FUNCTION_BLOCK Section1
  (* Standard: 61499-2 *)
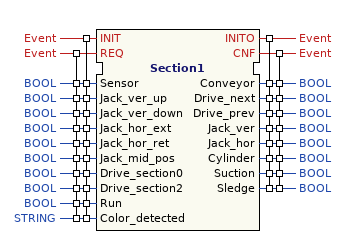
  EVENT_INPUT
    INIT WITH Sensor, Jack_ver_up, Jack_ver_down, Jack_hor_ext, Jack_hor_ret, Jack_mid_pos, Drive_section0, Drive_section2, Run, Color_detected;
    REQ WITH Sensor, Jack_ver_up, Jack_ver_down, Jack_hor_ext, Jack_hor_ret, Jack_mid_pos, Drive_section0, Drive_section2, Run, Color_detected;
  END_EVENT
  EVENT_OUTPUT
    INITO WITH Conveyor, Drive_next, Drive_prev, Jack_ver, Jack_hor, Cylinder, Suction, Sledge;
    CNF WITH Conveyor, Drive_next, Drive_prev, Jack_ver, Jack_hor, Cylinder, Suction, Sledge;
  END_EVENT
  VAR_INPUT
    Sensor : BOOL;
    Jack_ver_up : BOOL;
    Jack_ver_down : BOOL;
    Jack_hor_ext : BOOL;
    Jack_hor_ret : BOOL;
    Jack_mid_pos : BOOL;
    Drive_section0 : BOOL;
    Drive_section2 : BOOL;
    Run : BOOL;
    Color_detected : STRING;
  END_VAR
  VAR_OUTPUT
    Conveyor : BOOL;
    Drive_next : BOOL;
    Drive_prev : BOOL;
    Jack_ver : BOOL;
    Jack_hor : BOOL;
    Cylinder : BOOL;
    Suction : BOOL;
    Sledge : BOOL;
  END_VAR
  FBS
    FB3 : DisableConveyor;
    Section1Ctrl : Section1Ctrl;
    Jack1Ctrl : Jack1Ctrl;
  END_FBS
  EVENT_CONNECTIONS
    FB3.CNF TO CNF;
    INIT TO Section1Ctrl.INIT;
    Section1Ctrl.CNF TO Jack1Ctrl.REQ;
    REQ TO Jack1Ctrl.REQ;
    Section1Ctrl.INITO TO Jack1Ctrl.INIT;
    REQ TO Section1Ctrl.REQ;
    Jack1Ctrl.CNF TO Section1Ctrl.REQ;
    Section1Ctrl.CNF TO FB3.REQ;
    REQ TO FB3.REQ;
    Section1Ctrl.INITO TO FB3.INIT;
  END_CONNECTIONS
  DATA_CONNECTIONS
    Jack_ver_up TO Jack1Ctrl.JackVerUp;
    Jack_ver_down TO Jack1Ctrl.JackVerDown;
    Jack_hor_ext TO Jack1Ctrl.JackHorExt;
    Jack_hor_ret TO Jack1Ctrl.JackHorRet;
    Jack_mid_pos TO Jack1Ctrl.JackMidPos;
    Section1Ctrl.Jack1_removes TO Jack1Ctrl.Jack1_removes;
    Jack1Ctrl.ReadySIG TO Section1Ctrl.Jack1_finished;
    Sensor TO Section1Ctrl.Sensor;
    Section1Ctrl.Drive_next TO Drive_next;
    Section1Ctrl.Drive_prev TO Drive_prev;
    Section1Ctrl.Conveyor TO FB3.ConvIn;
    Run TO FB3.QI;
    FB3.ConvOut TO Conveyor;
    Color_detected TO Jack1Ctrl.Color_detected;
    Drive_section2 TO Section1Ctrl.Drive_section2;
    Drive_section0 TO Section1Ctrl.Drive_section0;
    Jack1Ctrl.JackVer TO Jack_ver;
    Jack1Ctrl.JackHor TO Jack_hor;
    Jack1Ctrl.Cylinder TO Cylinder;
    Jack1Ctrl.Suction TO Suction;
    Jack1Ctrl.Sledge TO Sledge;
  END_CONNECTIONS
END_FUNCTION_BLOCK
